(* Logix 5000 project; controller Uidaho_Factory vendor 1 type 14 code 165 rev 38.11; software revision 38.00; part 2 of 4 *)
(* tags used below, declared in another part *)
   ESTOP : BOOL;
   HBW_Start : DINT;
   MPO_Homing : BOOL;
   Start : DINT;
   Step : DINT[20];
   VGR_Step : DINT;
   X_Position : DINT;
   X_Position_Return : DINT;
   Y_Position : DINT;
   Y_Position_Drop_off : DINT;
   Y_Position_DropOff_At_Rack : DINT;
   Y_Position_Pick_Up : DINT;
   Y_Position_Return : DINT;
   Encoder_Counters_1X : COUNTER[10];
   Encoder_Counters_4X : COUNTER[10];
   HBW_PWM_Outputs : PWM_Out[20];
   I_O_Counter : COUNTER[20];
   Slot_1_Faulted : DINT;
   Slot_2_Faulted : DINT;
   Slot_3_Faulted : DINT;
   Slot_4_Faulted : DINT;
   Slot_5_Faulted : DINT;
   Slot_6_Faulted : DINT;
   Slot_7_Faulted : DINT;
   Slot_9_Faulted : DINT;
(* MainProgram, continued *)

ROUTINE HBW_Controller   (* ladder *)
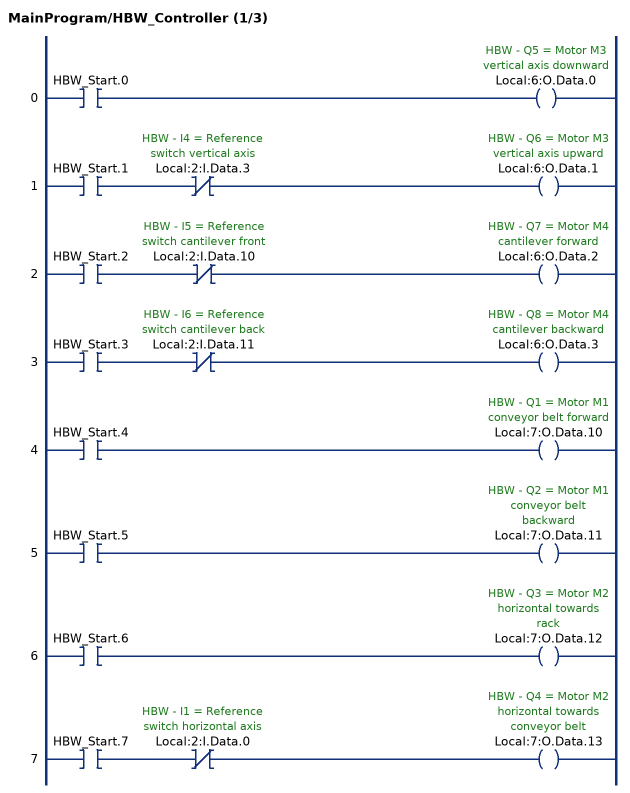
   0: XIC(HBW_Start.0)OTE(Local:6:O.Data.0);
   1: XIC(HBW_Start.1)XIO(Local:2:I.Data.3)OTE(Local:6:O.Data.1);
   2: XIC(HBW_Start.2)XIO(Local:2:I.Data.10)OTE(Local:6:O.Data.2);
   3: XIC(HBW_Start.3)XIO(Local:2:I.Data.11)OTE(Local:6:O.Data.3);
   4: XIC(HBW_Start.4)OTE(Local:7:O.Data.10);
   5: XIC(HBW_Start.5)OTE(Local:7:O.Data.11);
   6: XIC(HBW_Start.6)OTE(Local:7:O.Data.12);
   7: XIC(HBW_Start.7)XIO(Local:2:I.Data.0)OTE(Local:7:O.Data.13);
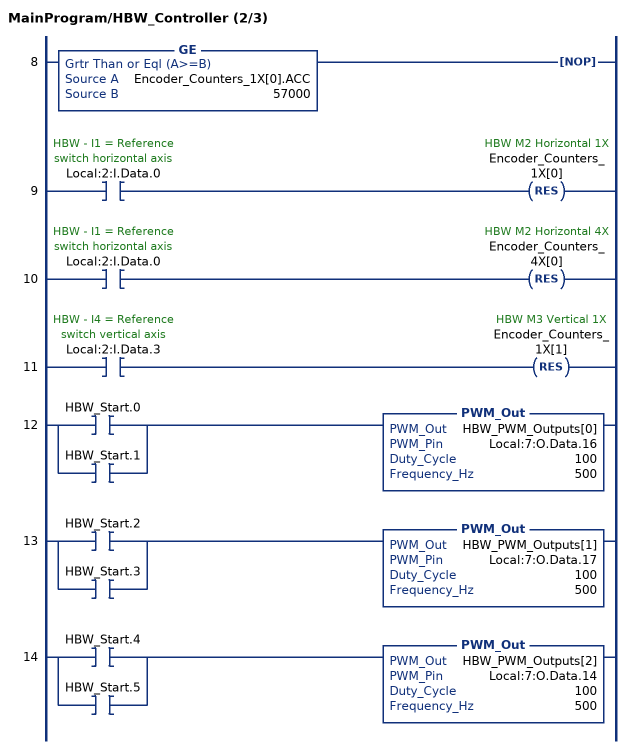
   8: GE(Encoder_Counters_1X[0].ACC,57000)NOP();
   9: XIC(Local:2:I.Data.0)RES(Encoder_Counters_1X[0]);
   10: XIC(Local:2:I.Data.0)RES(Encoder_Counters_4X[0]);
   11: XIC(Local:2:I.Data.3)RES(Encoder_Counters_1X[1]);
   12: [XIC(HBW_Start.0) ,XIC(HBW_Start.1) ]PWM_Out(HBW_PWM_Outputs[0],Local:7:O.Data.16,100,500);
   13: [XIC(HBW_Start.2) ,XIC(HBW_Start.3) ]PWM_Out(HBW_PWM_Outputs[1],Local:7:O.Data.17,100,500);
   14: [XIC(HBW_Start.4) ,XIC(HBW_Start.5) ]PWM_Out(HBW_PWM_Outputs[2],Local:7:O.Data.14,100,500);
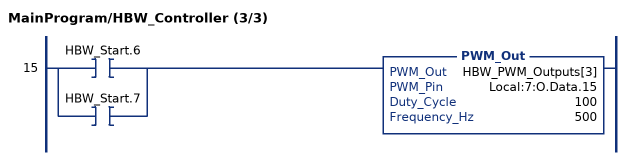
   15: [XIC(HBW_Start.6) ,XIC(HBW_Start.7) ]PWM_Out(HBW_PWM_Outputs[3],Local:7:O.Data.15,100,500);
END_ROUTINE

ROUTINE HBW_Sequencer   (* ladder *)
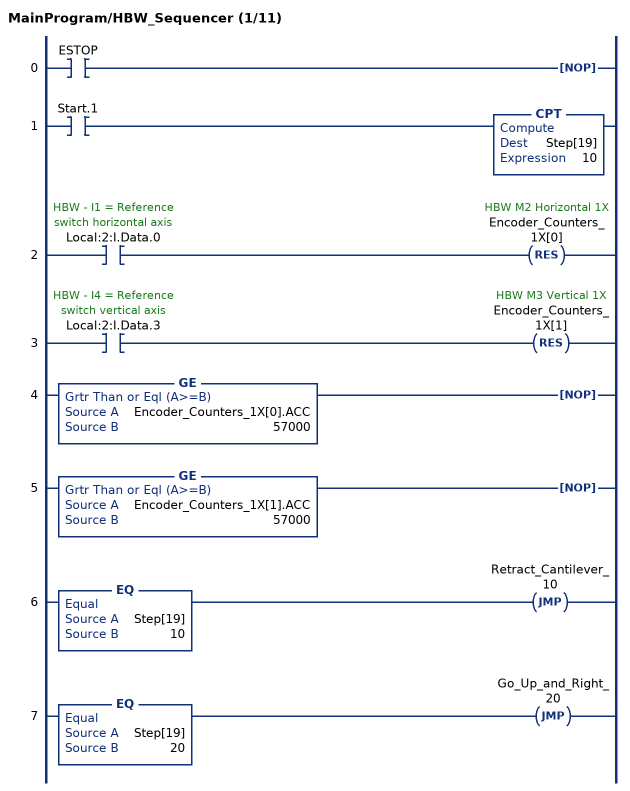
   0: XIC(ESTOP)NOP();
   1: XIC(Start.1)CPT(Step[19],10);
   2: XIC(Local:2:I.Data.0)RES(Encoder_Counters_1X[0]);
   3: XIC(Local:2:I.Data.3)RES(Encoder_Counters_1X[1]);
   4: GE(Encoder_Counters_1X[0].ACC,57000)NOP();
   5: GE(Encoder_Counters_1X[1].ACC,57000)NOP();
   6: EQ(Step[19],10)JMP(Retract_Cantilever_10);
   7: EQ(Step[19],20)JMP(Go_Up_and_Right_20);
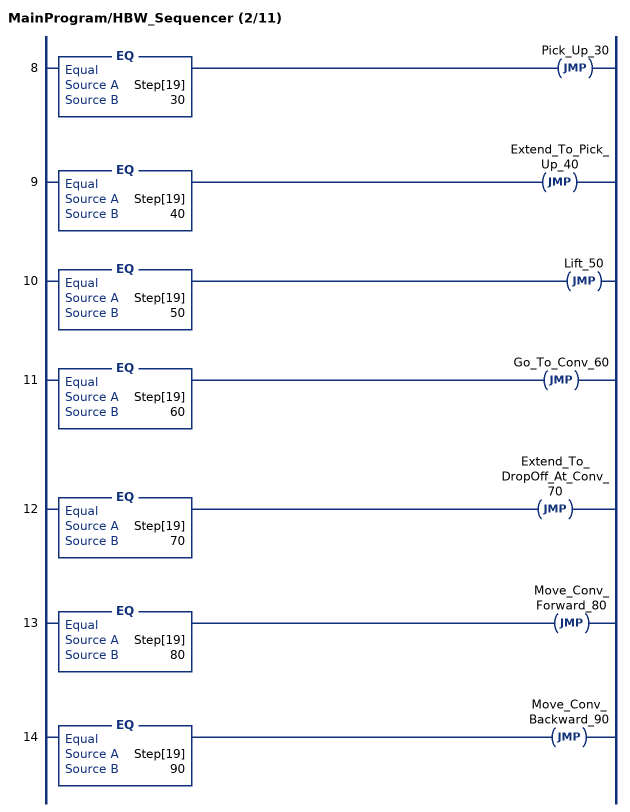
   8: EQ(Step[19],30)JMP(Pick_Up_30);
   9: EQ(Step[19],40)JMP(Extend_To_Pick_Up_40);
   10: EQ(Step[19],50)JMP(Lift_50);
   11: EQ(Step[19],60)JMP(Go_To_Conv_60);
   12: EQ(Step[19],70)JMP(Extend_To_DropOff_At_Conv_70);
   13: EQ(Step[19],80)JMP(Move_Conv_Forward_80);
   14: EQ(Step[19],90)JMP(Move_Conv_Backward_90);
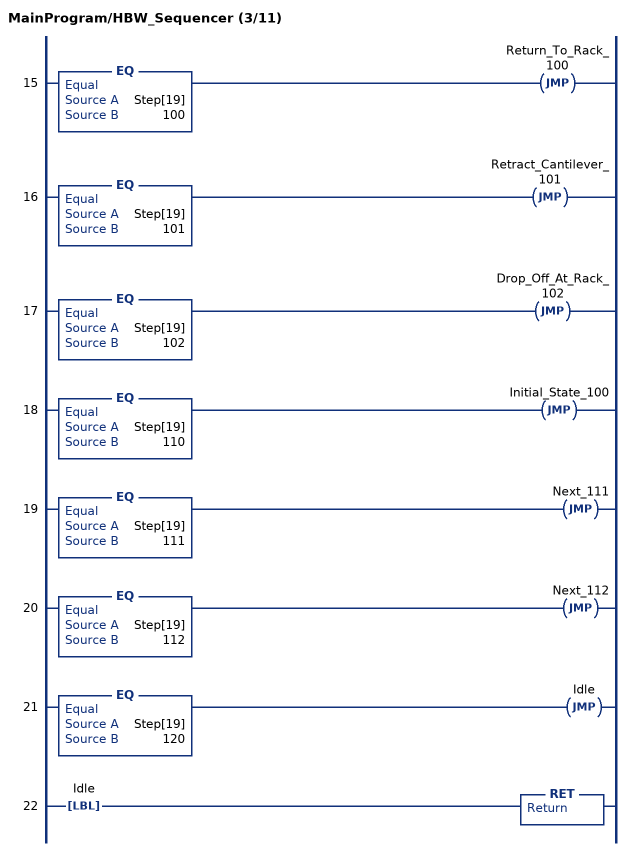
   15: EQ(Step[19],100)JMP(Return_To_Rack_100);
   16: EQ(Step[19],101)JMP(Retract_Cantilever_101);
   17: EQ(Step[19],102)JMP(Drop_Off_At_Rack_102);
   18: EQ(Step[19],110)JMP(Initial_State_100);
   19: EQ(Step[19],111)JMP(Next_111);
   20: EQ(Step[19],112)JMP(Next_112);
   21: EQ(Step[19],120)JMP(Idle);
   22: LBL(Idle)RET();
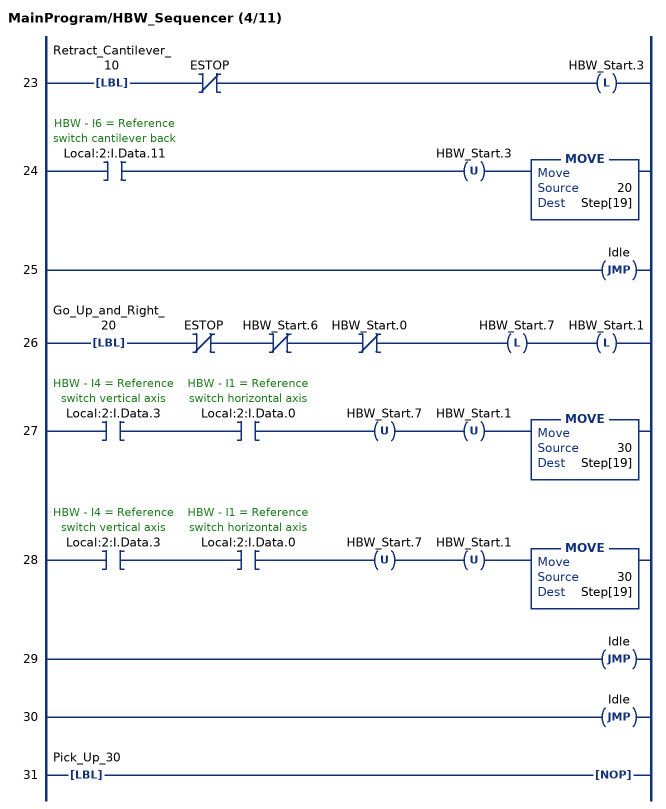
   23: LBL(Retract_Cantilever_10)XIO(ESTOP)OTL(HBW_Start.3);
   24: XIC(Local:2:I.Data.11)OTU(HBW_Start.3)MOVE(20,Step[19]);
   25: JMP(Idle);
   26: LBL(Go_Up_and_Right_20)XIO(ESTOP)XIO(HBW_Start.6)XIO(HBW_Start.0)OTL(HBW_Start.7)OTL(HBW_Start.1);
   27: XIC(Local:2:I.Data.3)XIC(Local:2:I.Data.0)OTU(HBW_Start.7)OTU(HBW_Start.1)MOVE(30,Step[19]);
   28: XIC(Local:2:I.Data.3)XIC(Local:2:I.Data.0)OTU(HBW_Start.7)OTU(HBW_Start.1)MOVE(30,Step[19]);
   29: JMP(Idle);
   30: JMP(Idle);
   31: LBL(Pick_Up_30)NOP();
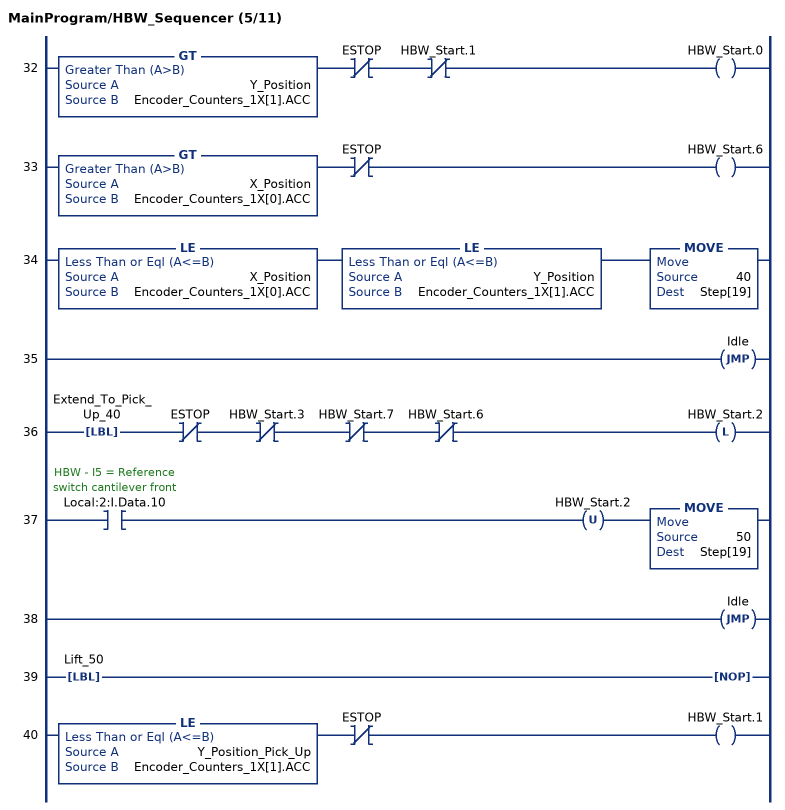
   32: GT(Y_Position,Encoder_Counters_1X[1].ACC)XIO(ESTOP)XIO(HBW_Start.1)OTE(HBW_Start.0);
   33: GT(X_Position,Encoder_Counters_1X[0].ACC)XIO(ESTOP)OTE(HBW_Start.6);
   34: LE(X_Position,Encoder_Counters_1X[0].ACC)LE(Y_Position,Encoder_Counters_1X[1].ACC)MOVE(40,Step[19]);
   35: JMP(Idle);
   36: LBL(Extend_To_Pick_Up_40)XIO(ESTOP)XIO(HBW_Start.3)XIO(HBW_Start.7)XIO(HBW_Start.6)OTL(HBW_Start.2);
   37: XIC(Local:2:I.Data.10)OTU(HBW_Start.2)MOVE(50,Step[19]);
   38: JMP(Idle);
   39: LBL(Lift_50)NOP();
   40: LE(Y_Position_Pick_Up,Encoder_Counters_1X[1].ACC)XIO(ESTOP)OTE(HBW_Start.1);
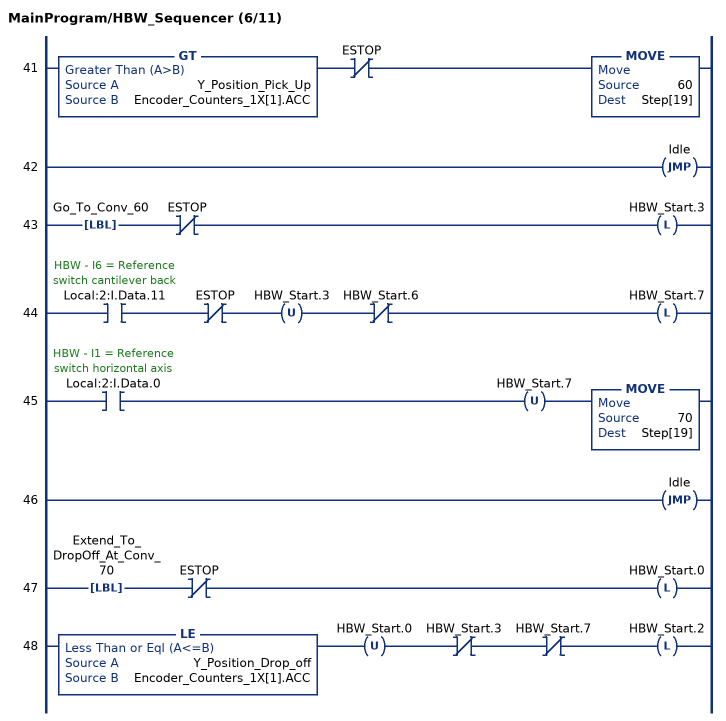
   41: GT(Y_Position_Pick_Up,Encoder_Counters_1X[1].ACC)XIO(ESTOP)MOVE(60,Step[19]);
   42: JMP(Idle);
   43: LBL(Go_To_Conv_60)XIO(ESTOP)OTL(HBW_Start.3);
   44: XIC(Local:2:I.Data.11)XIO(ESTOP)OTU(HBW_Start.3)XIO(HBW_Start.6)OTL(HBW_Start.7);
   45: XIC(Local:2:I.Data.0)OTU(HBW_Start.7)MOVE(70,Step[19]);
   46: JMP(Idle);
   47: LBL(Extend_To_DropOff_At_Conv_70)XIO(ESTOP)OTL(HBW_Start.0);
   48: LE(Y_Position_Drop_off,Encoder_Counters_1X[1].ACC)OTU(HBW_Start.0)XIO(HBW_Start.3)XIO(HBW_Start.7)OTL(HBW_Start.2);
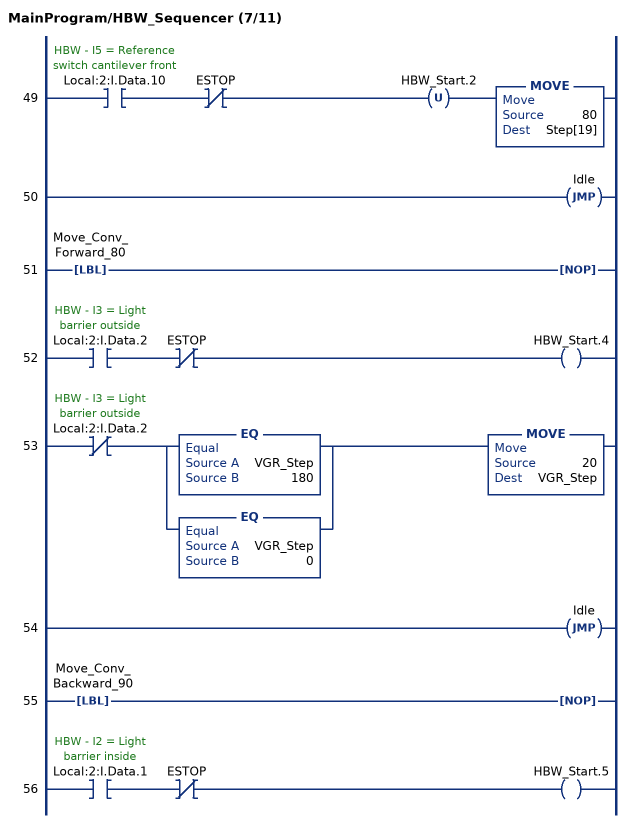
   49: XIC(Local:2:I.Data.10)XIO(ESTOP)OTU(HBW_Start.2)MOVE(80,Step[19]);
   50: JMP(Idle);
   51: LBL(Move_Conv_Forward_80)NOP();
   52: XIC(Local:2:I.Data.2)XIO(ESTOP)OTE(HBW_Start.4);
   53: XIO(Local:2:I.Data.2)[EQ(VGR_Step,180) ,EQ(VGR_Step,0) ]MOVE(20,VGR_Step);
   54: JMP(Idle);
   55: LBL(Move_Conv_Backward_90)NOP();
   56: XIC(Local:2:I.Data.1)XIO(ESTOP)OTE(HBW_Start.5);
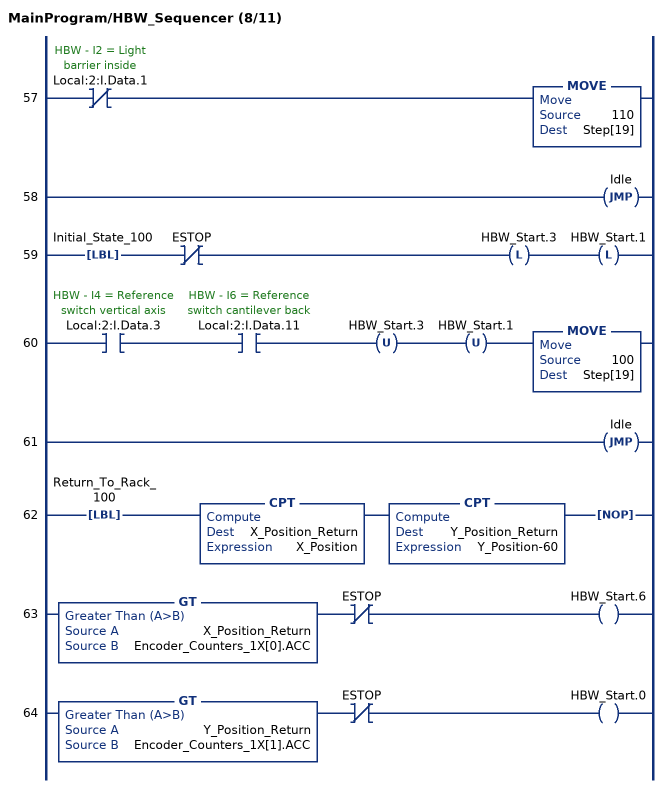
   57: XIO(Local:2:I.Data.1)MOVE(110,Step[19]);
   58: JMP(Idle);
   59: LBL(Initial_State_100)XIO(ESTOP)OTL(HBW_Start.3)OTL(HBW_Start.1);
   60: XIC(Local:2:I.Data.3)XIC(Local:2:I.Data.11)OTU(HBW_Start.3)OTU(HBW_Start.1)MOVE(100,Step[19]);
   61: JMP(Idle);
   62: LBL(Return_To_Rack_100)CPT(X_Position_Return,X_Position)CPT(Y_Position_Return,Y_Position-60)NOP();
   63: GT(X_Position_Return,Encoder_Counters_1X[0].ACC)XIO(ESTOP)OTE(HBW_Start.6);
   64: GT(Y_Position_Return,Encoder_Counters_1X[1].ACC)XIO(ESTOP)OTE(HBW_Start.0);
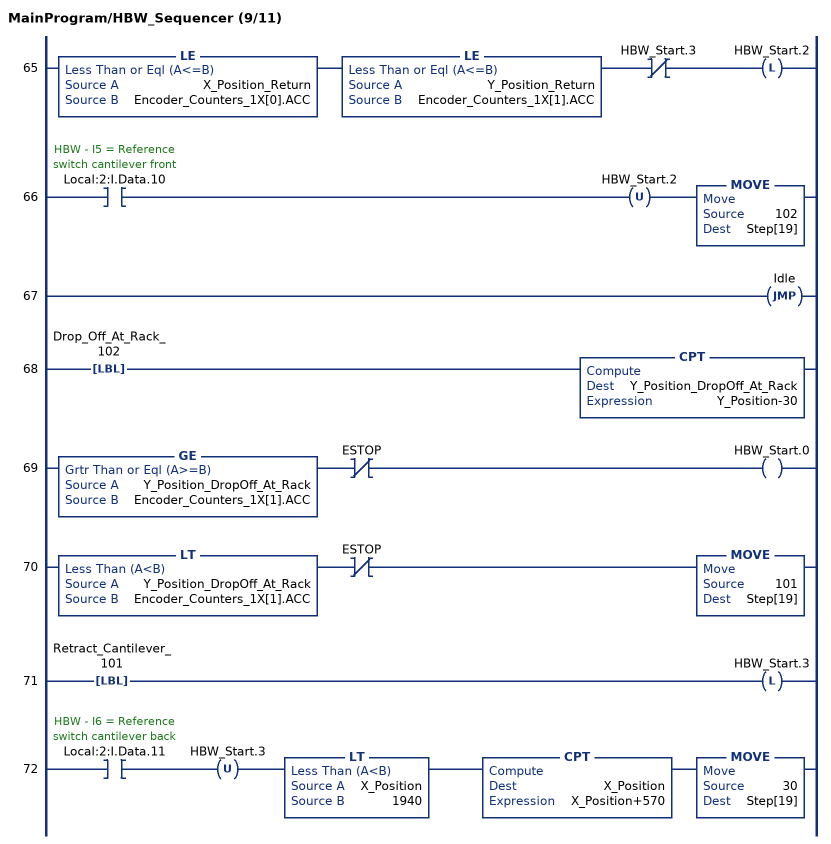
   65: LE(X_Position_Return,Encoder_Counters_1X[0].ACC)LE(Y_Position_Return,Encoder_Counters_1X[1].ACC)XIO(HBW_Start.3)OTL(HBW_Start.2);
   66: XIC(Local:2:I.Data.10)OTU(HBW_Start.2)MOVE(102,Step[19]);
   67: JMP(Idle);
   68: LBL(Drop_Off_At_Rack_102)CPT(Y_Position_DropOff_At_Rack,Y_Position-30);
   69: GE(Y_Position_DropOff_At_Rack,Encoder_Counters_1X[1].ACC)XIO(ESTOP)OTE(HBW_Start.0);
   70: LT(Y_Position_DropOff_At_Rack,Encoder_Counters_1X[1].ACC)XIO(ESTOP)MOVE(101,Step[19]);
   71: LBL(Retract_Cantilever_101)OTL(HBW_Start.3);
   72: XIC(Local:2:I.Data.11)OTU(HBW_Start.3)LT(X_Position,1940)CPT(X_Position,X_Position+570)MOVE(30,Step[19]);
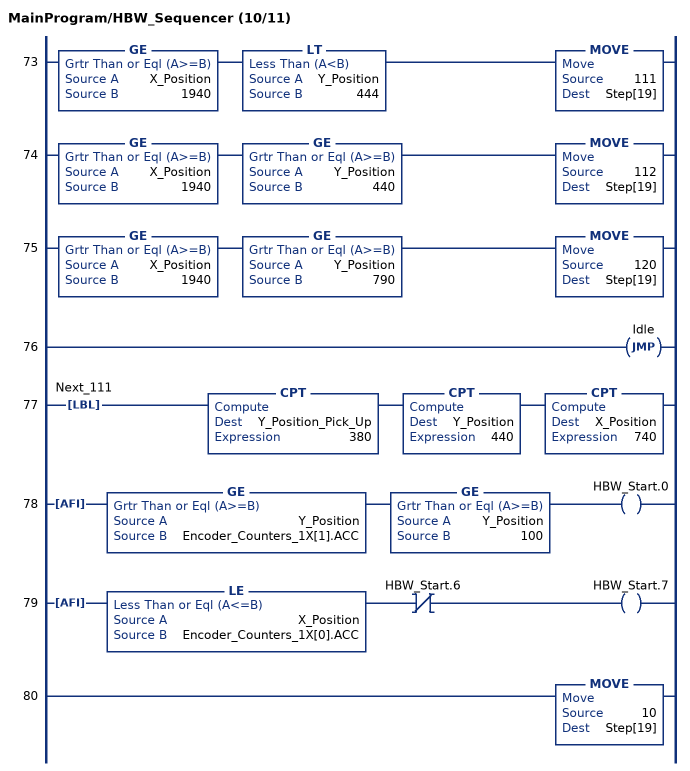
   73: GE(X_Position,1940)LT(Y_Position,444)MOVE(111,Step[19]);
   74: GE(X_Position,1940)GE(Y_Position,440)MOVE(112,Step[19]);
   75: GE(X_Position,1940)GE(Y_Position,790)MOVE(120,Step[19]);
   76: JMP(Idle);
   77: LBL(Next_111)CPT(Y_Position_Pick_Up,380)CPT(Y_Position,440)CPT(X_Position,740);
   78: AFI()GE(Y_Position,Encoder_Counters_1X[1].ACC)GE(Y_Position,100)OTE(HBW_Start.0);
   79: AFI()LE(X_Position,Encoder_Counters_1X[0].ACC)XIO(HBW_Start.6)OTE(HBW_Start.7);
   80: MOVE(10,Step[19]);
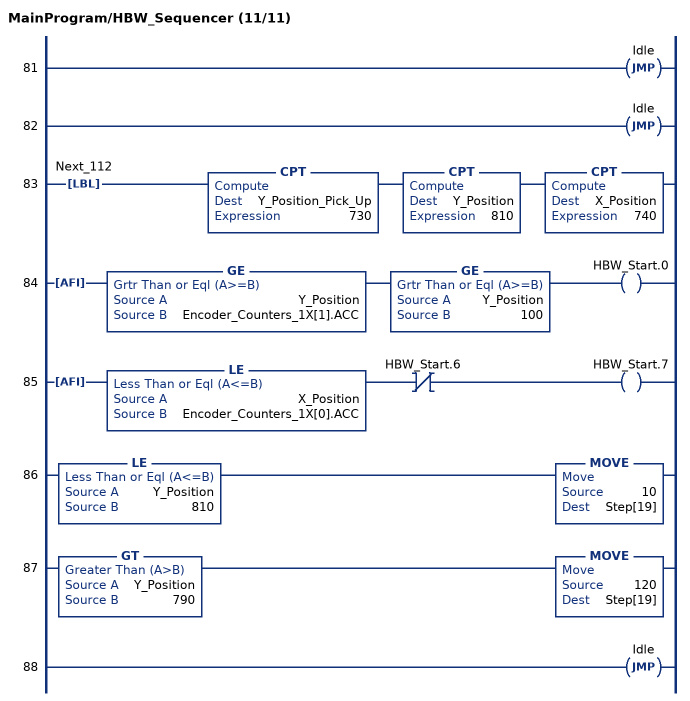
   81: JMP(Idle);
   82: JMP(Idle);
   83: LBL(Next_112)CPT(Y_Position_Pick_Up,730)CPT(Y_Position,810)CPT(X_Position,740);
   84: AFI()GE(Y_Position,Encoder_Counters_1X[1].ACC)GE(Y_Position,100)OTE(HBW_Start.0);
   85: AFI()LE(X_Position,Encoder_Counters_1X[0].ACC)XIO(HBW_Start.6)OTE(HBW_Start.7);
   86: LE(Y_Position,810)MOVE(10,Step[19]);
   87: GT(Y_Position,790)MOVE(120,Step[19]);
   88: JMP(Idle);
END_ROUTINE

ROUTINE MainRoutine   (* ladder *)
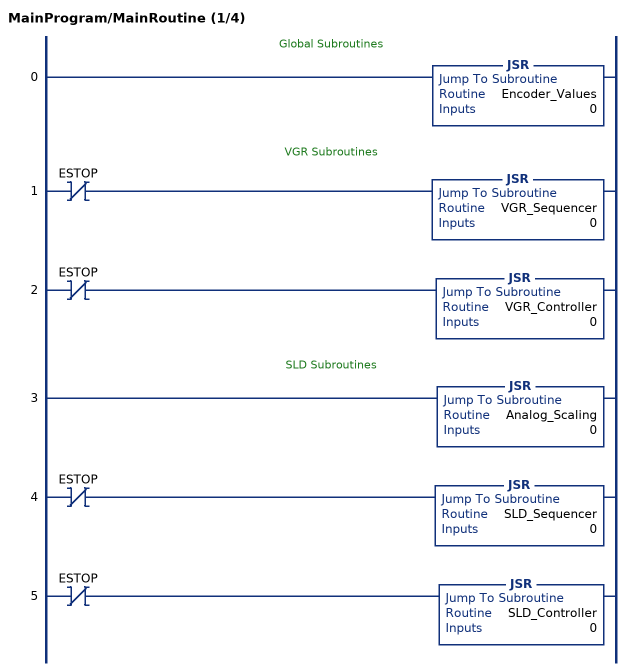
   // Global Subroutines
   0: JSR(Encoder_Values,0);
   // VGR Subroutines
   1: XIO(ESTOP)JSR(VGR_Sequencer,0);
   2: XIO(ESTOP)JSR(VGR_Controller,0);
   // SLD Subroutines
   3: JSR(Analog_Scaling,0);
   4: XIO(ESTOP)JSR(SLD_Sequencer,0);
   5: XIO(ESTOP)JSR(SLD_Controller,0);
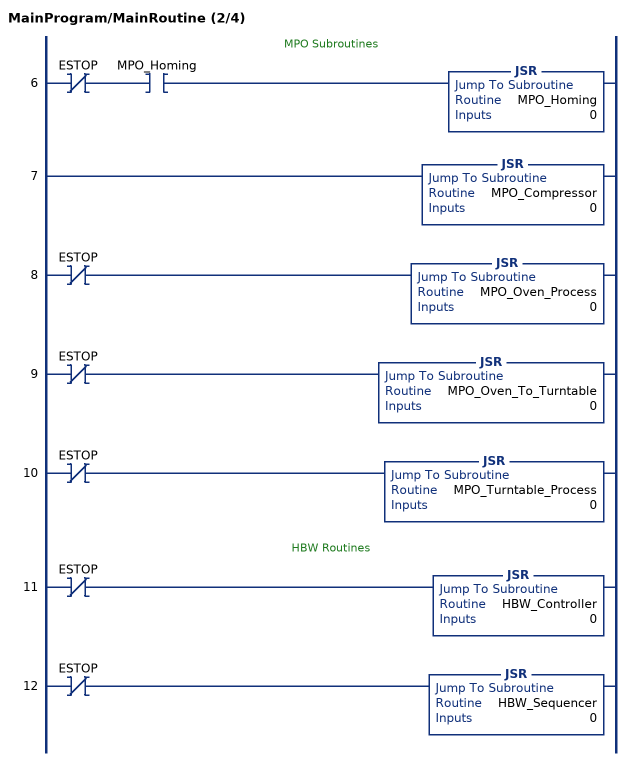
   // MPO Subroutines
   6: XIO(ESTOP)XIC(MPO_Homing)JSR(MPO_Homing,0);
   7: JSR(MPO_Compressor,0);
   8: XIO(ESTOP)JSR(MPO_Oven_Process,0);
   9: XIO(ESTOP)JSR(MPO_Oven_To_Turntable,0);
   10: XIO(ESTOP)JSR(MPO_Turntable_Process,0);
   // HBW Routines
   11: XIO(ESTOP)JSR(HBW_Controller,0);
   12: XIO(ESTOP)JSR(HBW_Sequencer,0);
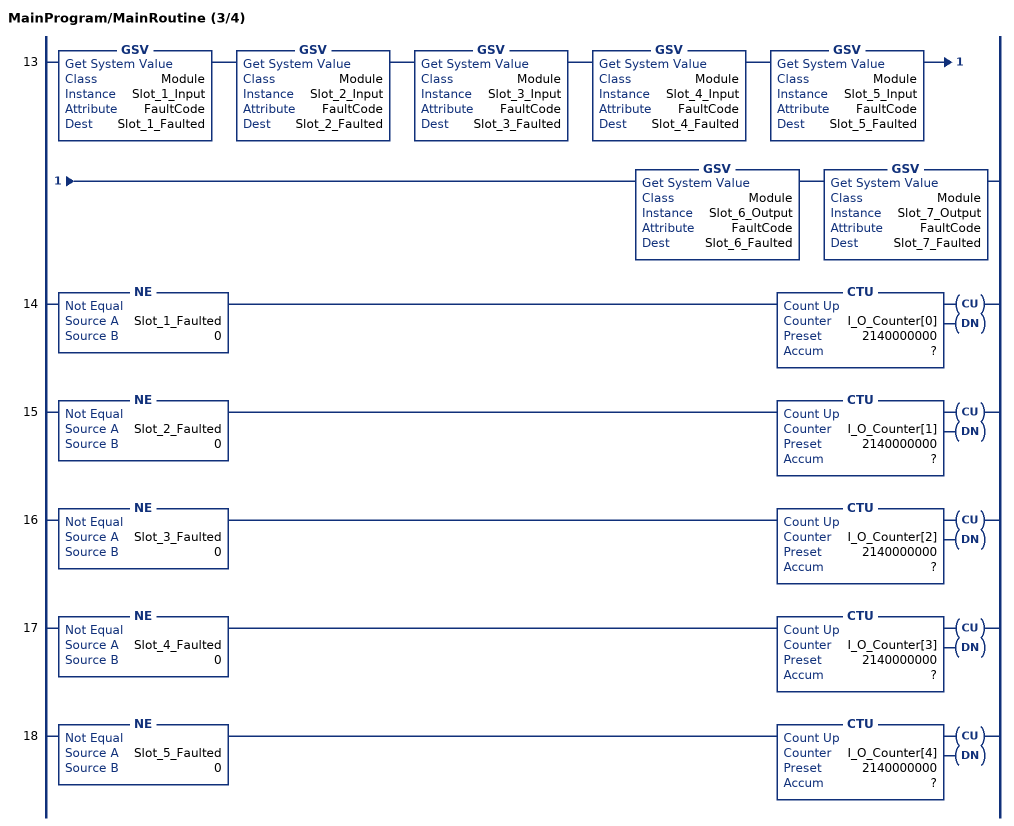
   13: GSV(Module,Slot_1_Input,FaultCode,Slot_1_Faulted)GSV(Module,Slot_2_Input,FaultCode,Slot_2_Faulted)GSV(Module,Slot_3_Input,FaultCode,Slot_3_Faulted)GSV(Module,Slot_4_Input,FaultCode,Slot_4_Faulted)GSV(Module,Slot_5_Input,FaultCode,Slot_5_Faulted)GSV(Module,Slot_6_Output,FaultCode,Slot_6_Faulted)GSV(Module,Slot_7_Output,FaultCode,Slot_7_Faulted);
   14: NE(Slot_1_Faulted,0)CTU(I_O_Counter[0],?,?);
   15: NE(Slot_2_Faulted,0)CTU(I_O_Counter[1],?,?);
   16: NE(Slot_3_Faulted,0)CTU(I_O_Counter[2],?,?);
   17: NE(Slot_4_Faulted,0)CTU(I_O_Counter[3],?,?);
   18: NE(Slot_5_Faulted,0)CTU(I_O_Counter[4],?,?);
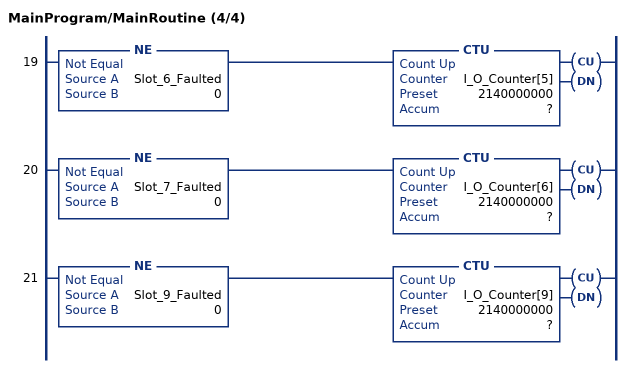
   19: NE(Slot_6_Faulted,0)CTU(I_O_Counter[5],?,?);
   20: NE(Slot_7_Faulted,0)CTU(I_O_Counter[6],?,?);
   21: NE(Slot_9_Faulted,0)CTU(I_O_Counter[9],?,?);
END_ROUTINE
